// TwinCAT 3 PLC project MqttTestPLC2
// ProgramVersion: 3.1.4023.0
// libraries:
//   ChainControllerLib, * (FactoryAutomation)
//   MqttFramework, * (FactoryAutomation)
//   StateMachineLib, * (FactoryAutomation)
//   StepWorkerLib, * (FactoryAutomation)
//   Tc2_Standard, * (Beckhoff Automation GmbH)
//   Tc2_System, * (Beckhoff Automation GmbH)
//   Tc3_Module, * (Beckhoff Automation GmbH)
// project tree:
//   / PlcTask.TcTTO
//   POUs/Basic/Conveyors/ BeltConveyor.TcPOU, Conveyor.TcPOU, PalletizerConveyor.TcPOU, RollerConveyor.TcPOU
//   POUs/Basic/Cylinder/ Cylinder.TcPOU
//   POUs/Basic/Elevator/ Elevator.TcPOU, PalletizerElevator.TcPOU
//   POUs/Basic/Sensor/ Sensor.TcPOU
//   POUs/HeavyModules/LineRegulator/ SM_LineRegulator.TcPOU
//   POUs/HeavyModules/TransferLine/ SM_TransferLine.TcPOU, TL_BUSY.TcDUT, TL_RollerConveyors.TcDUT
//   POUs/HeavyModules/TransferLine/StepChains/BeltConveyors/ SC_ACTUATOR_BeltConveyors.TcDUT, SC_BeltConveyors.TcPOU, SC_BUSY_BeltConveyors.TcDUT, SC_SENSOR_BeltConveyors.TcDUT
//   POUs/HeavyModules/TransferLine/StepChains/PostPalletizer/ SC_PostPalletizer.TcPOU
//   POUs/HeavyModules/TransferLine/StepChains/PrePalletizer/ SC_PrePalletizer.TcPOU
//   POUs/LightModules/PresenceDetector/ PresenceDetector.TcPOU
//   POUs/LightModules/Turntable/ Turntable.TcPOU
//   POUs/Main/ MAIN.TcPOU, MAIN_BUSY.TcDUT
//   POUs/MediumModules/Palletizer/ PAL_Busy.TcDUT, SM_Palletizer.TcPOU
//   POUs/MediumModules/Palletizer/StepChains/FirstFloor/ SC_BUSY_FirstFloor.TcDUT, SC_FirstFloor.TcPOU
//   POUs/MediumModules/Palletizer/StepChains/SecondFloor/ SC_BUSY_SecondFloor.TcDUT, SC_SecondFloor.TcPOU
//   VISUs/ Visu.TcPOU
// real-time tasks:
//   TASK PlcTask: cycle T#10ms, priority 21, ADS port 350

CONFIGURATION MqttTestPLC2
    RESOURCE PLC ON TwinCAT3
        TASK PlcTask(INTERVAL := T#10ms, PRIORITY := 21);
        PROGRAM MAIN WITH PlcTask : MAIN;
        PROGRAM ADS WITH PlcTask : ADS;
    END_RESOURCE
END_CONFIGURATION

// ---- POUs/HeavyModules/TransferLine/StepChains/BeltConveyors/SC_ACTUATOR_BeltConveyors.TcDUT

TYPE SC_ACTUATOR_BeltConveyors :
(
	eBeltConveyorEntrance := 1,
	eBeltConveyorUpwards,
	eMaxNumBeltConveyors
)UINT;
END_TYPE

// ---- POUs/HeavyModules/TransferLine/StepChains/BeltConveyors/SC_BUSY_BeltConveyors.TcDUT

TYPE SC_BUSY_BeltConveyors :
(
	eBusySCStart := 0,
	eStartEntranceConveyor,
	eStartUpwardsConveyor,
	eExecutePalletizer,
	eStopEntranceConveyor,
	eWaitForPalletizer,
	eSignalError
)UINT;
END_TYPE

// ---- POUs/HeavyModules/TransferLine/StepChains/BeltConveyors/SC_SENSOR_BeltConveyors.TcDUT

TYPE SC_SENSOR_BeltConveyors :
(
	eCounterSensor := 1,
	eBeltConveyorsMaxSensors
)UINT;
END_TYPE

// ---- POUs/HeavyModules/TransferLine/TL_BUSY.TcDUT

TYPE TL_BUSY :
(
	eTlStartUnits := 0,
	eTlCheckUnits,
	eTlSignalError
)UINT;
END_TYPE

// ---- POUs/HeavyModules/TransferLine/TL_RollerConveyors.TcDUT

TYPE TL_RollerConveyors :
(
	eRollerConveyorEntrance := 1,
	eRollerConveyorExit,
	eRollerConveyorPrePalletizer,
	eTlMaxNumRollerConveyors
)UINT;
END_TYPE

// ---- POUs/Main/MAIN_BUSY.TcDUT

TYPE MAIN_BUSY :
(
	eMainWaitStart := 0
);
END_TYPE

// ---- POUs/MediumModules/Palletizer/PAL_Busy.TcDUT

TYPE PAL_Busy :
(
	ePALStart := 0
	
	
);
END_TYPE

// ---- POUs/MediumModules/Palletizer/StepChains/FirstFloor/SC_BUSY_FirstFloor.TcDUT

TYPE SC_BUSY_FirstFloor :
(
	enum_member := 0
);
END_TYPE

// ---- POUs/MediumModules/Palletizer/StepChains/SecondFloor/SC_BUSY_SecondFloor.TcDUT

TYPE SC_BUSY_SecondFloor :
(
	eSecondFloorStart := 0,
	eActivateTurn,
	eActivateBeltForw,
	eWaitForPackages,
	ePushPackages,
	eRetractPusher,
	eClamp,
	eRetractClamper,
	eWaitForPallet,
	eOpenPlate,
	eClosePlate,
	eElevatorUp,
	eElevatorDown,
	eStartChains,
	eStopChains,
	eWaitForFirstFloor,
	eSyncWithFirstFloor,
	eSecondFloorDone
);
END_TYPE

// ---- POUs/Main/MAIN.TcPOU
PROGRAM MAIN
VAR
 
 fbLineRegulator : SM_LineRegulator;
 fbSymbolPathStorage : SymbolPathStorage;

END_VAR

fbLineRegulator(
	 sSubscription1 := 'TL1Synch',
	 sSubscription2 := 'TL2Synch',
	 sSubscription3 := 'TL3Synch'
);

END_PROGRAM

// ---- POUs/HeavyModules/LineRegulator/SM_LineRegulator.TcPOU
FUNCTION_BLOCK SM_LineRegulator EXTENDS StateMachine
VAR_INPUT
	 sSubscription1 : STRING(8);
	 sSubscription2 : STRING(8);
	 sSubscription3 : STRING(8);
END_VAR
VAR_OUTPUT
END_VAR
VAR
	fbTurntable : Turntable;

	aRollerConveyors : ARRAY[1..3] OF RollerConveyor;
	fbRollerConveyorExit : RollerConveyor;
	fbReadyStepWorker : FB_StepWorker;
	fbBusyStepWorker : FB_StepWorker;
	fbInitStepWorker : FB_StepWorker;
	
	messageIndex : UINT;
	stMqttPayload : ST_MqttPayload;
	aSubscriptions : ARRAY[1..3] OF STRING(8);
	uiSubscriptionsCycler : UINT := 1;
END_VAR

SUPER^();
fbTurntable();
aRollerConveyors[1]();
aRollerConveyors[3]();

METHOD PROTECTED   Busy : BOOL
VAR_INPUT
END_VAR
fbBusyStepWorker();
CASE fbBusyStepWorker.uiStep OF

	0:
	
		aRollerConveyors[uiSubscriptionsCycler].On();
		CASE uiSubscriptionsCycler OF
		
			1:
				fbTurntable.RollMinus();
				fbTurntable.Turn();
			
			2:
				fbTurntable.RollPlus();
			
			3:
				fbTurntable.RollPlus();
				fbTurntable.Turn();
		END_CASE
		
		fbBusyStepWorker
			.mAddCondition(itfStepCondition := fbTurntable.fbBackLimit.getSignal)
			.mNextStep(10);
			
	10:
	
		aRollerConveyors[uiSubscriptionsCycler].Off();
		CASE uiSubscriptionsCycler OF
		
			1:
				fbTurntable.StopRolling();			
				fbTurntable.UnTurn();
				fbBusyStepWorker
					.mSetTimer(T#2S)
					.mNextStep(20);
			
			2:
				fbBusyStepWorker.mNextStep(30);
			
			3:
				fbTurntable.StopRolling();
				fbTurntable.UnTurn();
				fbBusyStepWorker
					.mSetTimer(T#2S)
					.mNextStep(20);
		END_CASE
		
	20:
	
		fbTurntable.RollPlus();
		fbRollerConveyorExit.On();
		fbBusyStepWorker
			.mSetTimer(T#10S)
			.mNextStep(30);
	30:	
	
		IF NOT fbTurntable.fbBackLimit.bSignal
			AND NOT fbTurntable.fbFrontLimit.bSignal
		THEN
			fbRollerConveyorExit.Off();
			fbBusyStepWorker
				.mSetTimer(T#1S)
				.mNextStep(40);
		END_IF
		
	40:
	
		fbBusyStepWorker.mNextStep(0);
		Done();
		
	
END_CASE
END_METHOD

METHOD PROTECTED  Error : BOOL
VAR_INPUT
END_VAR
END_METHOD

METHOD PROTECTED  Idle : BOOL
VAR_INPUT
END_VAR
END_METHOD

METHOD PROTECTED  Init : BOOL
VAR_INPUT
END_VAR
fbInitStepWorker();
CASE fbInitStepWorker.uiStep OF

	0: 
	
		IF ADS.fbAdsConnector.isConnected
		THEN
			fbInitStepWorker.mNextStep(10);
		END_IF
		
	10:
	
		IF ADS.fbMqttClient.Subscribe(sSubscription1)
		THEN			
			fbInitStepWorker.mNextStep(20);
		END_IF
		
	20:
	
		IF ADS.fbMqttClient.Subscribe(sSubscription2)
		THEN			
			fbInitStepWorker.mNextStep(30);
		END_IF
		
	30:
		
		IF ADS.fbMqttClient.Subscribe(sSubscription3)
		THEN		
			aSubscriptions[1] := sSubscription1;
			aSubscriptions[2] := sSubscription2;
			aSubscriptions[3] := sSubscription3;
			Start();
		END_IF		
		
END_CASE
END_METHOD

METHOD PROTECTED  Prepare : BOOL
VAR_INPUT
END_VAR
END_METHOD

METHOD PROTECTED  Ready : BOOL
VAR_INPUT
END_VAR
VAR
	
END_VAR
fbReadyStepWorker();


CASE fbReadyStepWorker.uiStep OF

	0: 
		IF NOT fbTurntable.bBackLimit
			AND NOT fbTurntable.bFrontLimit
		THEN
			fbReadyStepWorker.mNextStep(10);
		END_IF
		
	10:
	
		IF uiSubscriptionsCycler = 3
		THEN
			uiSubscriptionsCycler := 1;
		ELSE
			uiSubscriptionsCycler := uiSubscriptionsCycler + 1;
		END_IF
		
		messageIndex := ADS.fbMqttClient.isNewMessage(aSubscriptions[uiSubscriptionsCycler]);
		IF messageIndex > 0
		THEN
			stMqttPayload := Ads.fbMqttClient.getNewMessage(messageIndex);
			fbReadyStepWorker.mNextStep(20);
		END_IF
		
	20:	
		Ads.fbMqttClient.Publish(aSubscriptions[uiSubscriptionsCycler],stMqttPayload);
		fbReadyStepWorker.mNextStep(0);
		Execute();
		
END_CASE
END_METHOD

METHOD PROTECTED  Waiting : BOOL
VAR_INPUT
END_VAR
END_METHOD

END_FUNCTION_BLOCK

// ---- POUs/LightModules/Turntable/Turntable.TcPOU
FUNCTION_BLOCK Turntable
VAR_INPUT



END_VAR
VAR_OUTPUT

	bTurn 		: BOOL;
	bRollPlus	: BOOL;
	bRollMinus 	: BOOL;
	bFrontLimit : BOOL;
	bBackLimit	: BOOL;
	
END_VAR
VAR

	fbFrontLimit : Sensor;
	fbBackLimit : Sensor;
	
	fbTurn : BoolOut;
	fbRollPlus : BoolOut;
	fbRollMinus : BoolOut;
	
END_VAR

fbFrontLimit();
fbBackLimit();

bTurn := fbTurn.getValue;
bRollPlus := fbRollPlus.getValue;
bRollMinus := fbRollMinus.getValue;
bFrontLimit := fbFrontLimit.bSignal;
bBackLimit	:= fbBackLimit.bSignal;

METHOD RollMinus : BOOL
VAR_INPUT
END_VAR
fbRollMinus.setValue := TRUE;
fbRollPlus.setValue := FALSE;
END_METHOD

METHOD RollPlus : BOOL
VAR_INPUT
END_VAR
fbRollPlus.setValue := TRUE;
fbRollMinus.setValue := FALSE;
END_METHOD

METHOD StopRolling : BOOL
VAR_INPUT
END_VAR
fbRollMinus.setValue := FALSE;
fbRollPlus.setValue := FALSE;
END_METHOD

METHOD Turn : BOOL
VAR_INPUT
END_VAR
fbTurn.setValue := TRUE;
END_METHOD

METHOD Unturn : BOOL
VAR_INPUT
END_VAR
fbTurn.setValue := FALSE;
END_METHOD

END_FUNCTION_BLOCK

// ---- POUs/Basic/Sensor/Sensor.TcPOU
FUNCTION_BLOCK Sensor
VAR_INPUT
END_VAR
VAR_OUTPUT
	bSignal  : BOOL;
END_VAR
VAR
	fbSignal : BoolIn;
END_VAR

bSignal := fbSignal.getValue;

PROPERTY getSignal : I_StepCondition
GET
getSignal := fbSignal;
END_GET
END_PROPERTY

END_FUNCTION_BLOCK

// ---- POUs/Basic/Conveyors/RollerConveyor.TcPOU
FUNCTION_BLOCK RollerConveyor EXTENDS Conveyor
VAR_INPUT
END_VAR
VAR_OUTPUT
END_VAR
VAR
END_VAR

Super^();

END_FUNCTION_BLOCK

// ---- POUs/Basic/Conveyors/Conveyor.TcPOU
FUNCTION_BLOCK Conveyor 
VAR_INPUT
END_VAR

VAR_OUTPUT
	bStart  : BOOL;
END_VAR
VAR
	fbStart : BoolOut;
END_VAR

bStart := fbStart.getValue;

PROPERTY getStart : I_StepCondition
GET
getStart := fbStart;
END_GET
END_PROPERTY

METHOD Off : BOOL
VAR_INPUT
END_VAR
fbStart.setValue := FALSE;
END_METHOD

METHOD On : BOOL
VAR_INPUT
END_VAR
fbStart.setValue := TRUE;
END_METHOD

END_FUNCTION_BLOCK

// ---- POUs/Basic/Conveyors/BeltConveyor.TcPOU
FUNCTION_BLOCK BeltConveyor EXTENDS Conveyor
VAR_INPUT
END_VAR
VAR_OUTPUT
END_VAR
VAR
END_VAR

Super^();

END_FUNCTION_BLOCK

// ---- POUs/Basic/Conveyors/PalletizerConveyor.TcPOU
FUNCTION_BLOCK PalletizerConveyor EXTENDS Conveyor
VAR_INPUT
END_VAR
VAR_OUTPUT
	bStartBackward : BOOL;
END_VAR
VAR	
	fbStartBackward : BoolOut;
END_VAR

SUPER^();
bStartBackward := fbStartBackward.getValue;

PROPERTY getStartBackward : I_StepCondition
GET
getStartBackward := fbStartBackward;
END_GET
END_PROPERTY

END_FUNCTION_BLOCK

// ---- POUs/Basic/Cylinder/Cylinder.TcPOU
FUNCTION_BLOCK Cylinder 
VAR_INPUT
END_VAR
VAR_OUTPUT
	bExtended : BOOL;
	bExtend : BOOL;
END_VAR
VAR
	fbExtendedSignal : BoolIn;
	fbExtend : BoolOut;
END_VAR

bExtended := fbExtendedSignal.getValue;
bExtend := fbExtend.getValue;

METHOD Extend : BOOL
VAR_INPUT
END_VAR
fbExtend.setValue := TRUE;
END_METHOD

PROPERTY getExtend : I_StepCondition
GET
getExtend := fbExtend;
END_GET
END_PROPERTY

METHOD Retract : BOOL
VAR_INPUT
END_VAR
fbExtend.setValue := FALSE;
END_METHOD

END_FUNCTION_BLOCK

// ---- POUs/Basic/Elevator/Elevator.TcPOU
FUNCTION_BLOCK Elevator
VAR_INPUT
END_VAR
VAR_OUTPUT
END_VAR
VAR
END_VAR

END_FUNCTION_BLOCK

// ---- POUs/Basic/Elevator/PalletizerElevator.TcPOU
FUNCTION_BLOCK PalletizerElevator EXTENDS Elevator
VAR_INPUT
END_VAR
VAR_OUTPUT
	isMoving : BOOL;
END_VAR
VAR
	fbElevatorMoving : Sensor;
	fbElevatorUp : BoolOut;
	fbElevatorDown : BoolOut;
	fbElevatorToLimit : BoolOut;
END_VAR

isMoving := fbElevatorMoving.bSignal;

PROPERTY getElevatorMoving : I_StepCondition
GET
getElevatorMoving := fbElevatorMoving.getSignal;
END_GET
END_PROPERTY

METHOD MoveDown : BOOL
VAR_INPUT
END_VAR
fbElevatorDown.setValue := TRUE;
fbElevatorUp.setValue := FALSE;

fbElevatorToLimit.setValue := TRUE;
END_METHOD

METHOD MoveUp : BOOL
VAR_INPUT
END_VAR
fbElevatorUp.setValue := TRUE;
fbElevatorDown.setValue := FALSE;

fbElevatorToLimit.setValue := TRUE;
END_METHOD

END_FUNCTION_BLOCK

// ---- POUs/HeavyModules/TransferLine/SM_TransferLine.TcPOU
FUNCTION_BLOCK SM_TransferLine EXTENDS StateMachine
VAR_INPUT CONSTANT
	sTLMqttName : STRING(8);
END_VAR
VAR_OUTPUT
END_VAR
VAR
	
	aRollerConveyors : ARRAY[1..3] OF RollerConveyor;
	fbChainController : FB_ChainController;
	
	fbPalletizer : SM_Palletizer;
	fbStepWorkerReady : FB_StepWorker;
	fbStepWorkerBusy : FB_StepWorker;

	scBeltConveyors : 
		SC_BeltConveyors := 
		(
			sChainName  := 'scBeltConveyors',
			rChainController := fbChainController
		);
		
	scPostPalletizer : 
		SC_PostPalletizer := 
		(
			sChainName  := 'scPostPalletizer',
			rChainController := fbChainController
		);
		
	scPrePalletizer : 
		SC_PrePalletizer := 
		(
			sChainName  := 'scPrePalletizer',
			rChainController := fbChainController
		);
 
	uiPackageCounter : UINT;
	i : UINT;
	bPackageOnTheWay : BOOL;
	
END_VAR

SUPER^();
fbPalletizer(ioChainController := fbChainController);
scBeltConveyors(bAllPartsPresent := fbPalletizer.bAllPartsPresent);
scPrePalletizer();
scPrePalletizer.bPalletizerRequest := fbPalletizer.scFirstFloor.bPalletizerRequest;
fbPalletizer.scFirstFloor.bIncomingPallet := scPrePalletizer.bSentToPalletizer;
scPostPalletizer(sTLMqttName := sTLMqttName);

METHOD PROTECTED Busy : BOOL
VAR_INPUT
END_VAR
CASE fbStepWorkerBusy.uiStep OF
	eTlStartUnits:
		scBeltConveyors.bExecute := TRUE;
		scPrePalletizer.bExecute := TRUE;
		scPostPalletizer.bExecute := TRUE;
		fbPalletizer.bExecute := TRUE;
		fbStepWorkerBusy.mNextStep(eTlCheckUnits);
	eTlCheckUnits:
		IF scBeltConveyors.eStateMachine = E_StateMachine.eError
		THEN
			fbStepWorkerBusy.mNextStep(eTlSignalError);
		END_IF
	eTlSignalError:
		Fault();
END_CASE
END_METHOD

METHOD PROTECTED  Error : BOOL
VAR_INPUT
END_VAR
END_METHOD

METHOD PROTECTED  Idle : BOOL
VAR_INPUT
END_VAR
Start();
END_METHOD

METHOD PROTECTED  Init : BOOL
VAR_INPUT
END_VAR
fbChainController
	.addChain(itfChain := scBeltConveyors)
	.addChain(itfChain := scPostPalletizer)
	.addChain(itfChain := scPrePalletizer);
	
	
Start();
END_METHOD

METHOD PROTECTED  Prepare : BOOL
VAR_INPUT
END_VAR
END_METHOD

METHOD PROTECTED  Ready : BOOL
VAR_INPUT
END_VAR
END_METHOD

METHOD PROTECTED  Waiting : BOOL
VAR_INPUT
END_VAR
END_METHOD

END_FUNCTION_BLOCK

// ---- POUs/MediumModules/Palletizer/SM_Palletizer.TcPOU
FUNCTION_BLOCK SM_Palletizer EXTENDS StateMachine
VAR_INPUT
	bExecute : BOOL;
	scFirstFloor : SC_FirstFloor;	
	scSecondFloor : SC_SecondFloor;
END_VAR
VAR_IN_OUT
	ioChainController : FB_ChainController;
END_VAR
VAR_OUTPUT
	
	bAllPartsPresent: BOOL;	
	
END_VAR
VAR

	fbDoneCycle : BoolOut;
	fbStepWorkerBusy : FB_StepWorker;
	
	
END_VAR

SUPER^();
scFirstFloor(bExecute := bExecute);
scSecondFloor(bExecute := bExecute);

bAllPartsPresent := scSecondFloor.bAllPartsPresent;
scSecondFloor.bPlateOpen := scFirstFloor.bPlateOpen;

METHOD PROTECTED   Busy : BOOL
VAR_INPUT
END_VAR
scFirstFloor(bExecute := TRUE);
scSecondFloor(bExecute := TRUE);
END_METHOD

METHOD PROTECTED  Error : BOOL
VAR_INPUT
END_VAR
END_METHOD

PROPERTY getDoneCycle : I_StepCondition
GET
getDoneCycle := fbDoneCycle;
END_GET
END_PROPERTY

METHOD PROTECTED  Idle : BOOL
VAR_INPUT
END_VAR
Start();
END_METHOD

METHOD PROTECTED  Init : BOOL
VAR_INPUT
END_VAR
ioChainController
	.addChain(itfChain := scFirstFloor)
	.addChain(itfChain := scSecondFloor);
	
scFirstFloor(
	sChainName := 'scFirstFloor',
	rChainController := ioChainController
);
scSecondFloor(
	sChainName := 'scSecondFloor',
	rChainController := ioChainController
);
Start();
END_METHOD

METHOD PROTECTED  Prepare : BOOL
VAR_INPUT
END_VAR
END_METHOD

METHOD PROTECTED  Ready : BOOL
VAR_INPUT
END_VAR
END_METHOD

METHOD PROTECTED  Waiting : BOOL
VAR_INPUT
END_VAR
END_METHOD

END_FUNCTION_BLOCK

// ---- POUs/MediumModules/Palletizer/StepChains/FirstFloor/SC_FirstFloor.TcPOU
FUNCTION_BLOCK SC_FirstFloor EXTENDS FB_Chain
VAR_INPUT
	bExecute : BOOL;
	bIncomingPallet : BOOL;
	bPostPalletizerRequestGranted : BOOL;
END_VAR
VAR_OUTPUT
	bPlateOpen : BOOL;
	bPalletizerRequest : BOOL;
	bSentToPostPalletizer : BOOL;
	bPostPalletizerDeliveryRequest : BOOL;
END_VAR
VAR
	fbPallChainConveyor : PalletizerConveyor;
	fbPallElevator : PalletizerElevator;
	fbPlateCyl : Cylinder;
	fbPlateLimitSen : Sensor;
	fbElevatorFrontLimit : Sensor;
	fbElevatorBackLimit : Sensor;
END_VAR

SUPER^();
bPlateOpen := fbPlateCyl.bExtended;
fbPallChainConveyor();
fbPallElevator();
fbPlateCyl();
fbPlateLimitSen();

METHOD PROTECTED   Busy : BOOL
VAR_INPUT
END_VAR

		
fbStepWorkerBusy();
CASE fbStepWorkerBusy.uiStep OF
	
	0: 
		fbPallChainConveyor.On();
		fbStepWorkerBusy
			.mAddCondition(itfStepCondition := fbElevatorBackLimit.getSignal)
			.mAddCondition(itfStepCOndition := fbElevatorFrontLimit.getSignal)
			.mNextStep(10);
			
	10: 
	
		fbPallChainConveyor.Off();
		bPalletizerRequest := FALSE;
		IF rChainController
			.releaseCheck(THIS^)
			.releaseFromChain(sChainReleasing := 'scSecondFloor', THIS^)
			.releaseResult(THIS^) 
		THEN
			fbStepWorkerBusy.mNextStep(20);
		END_IF

	20:
	
		fbPallElevator.MoveUp();
		fbStepWorkerBusy
			.mSetTimer(T#1S)
			.mNextStep(30);
			
	30:
	
		IF NOT fbPallElevator.isMoving
		THEN
			fbStepWorkerBusy
				.mSetTimer(tTime := T#2S)
				.mNextStep(40);
		END_IF
		
	40:
	
		fbPlateCyl.Extend();
		fbStepWorkerBusy
			.mSetTimer(T#2S)
			.mNextStep(45);
	
	45:	
		rChainController.releaseForChain('scSecondFloor', THIS^);	
		fbPallElevator.MoveDown();		
		fbStepWorkerBusy
			.mSetTimer(T#2S)
			.mNextStep(50);
	50:
	
		IF NOT fbPallElevator.isMoving
		THEN
			rChainController.releaseForChain('scPostPalletizer', THIS^);
			fbStepWorkerBusy.mNextStep(60);
		END_IF
	
		
	60:
	
		fbPlateCyl.Retract();
		fbStepWorkerBusy.mNextStep(100);
	
	100:
	
		IF rChainController
			.releaseCheck(THIS^)
			.releaseFromChain(sChainReleasing := 'scPostPalletizer', THIS^)
			.releaseResult(THIS^) 
		THEN

			fbPallChainConveyor.On();
			fbStepWorkerBusy.mNextStep(105);
			
		END_IF

	105:
		fbStepWorkerBusy
				.mSetTimer(T#2s)
				.mNextStep(110);
	110:		
		
		IF NOT fbElevatorBackLimit.bSignal
			AND NOT fbElevatorFrontLimit.bSignal
		THEN
		
			Done();
			fbPallChainConveyor.Off();
			fbStepWorkerBusy.mNextStep(0);
		END_IF

END_CASE
END_METHOD

METHOD PROTECTED  Error : BOOL
VAR_INPUT
END_VAR
END_METHOD

METHOD PROTECTED  Idle : BOOL
VAR_INPUT
END_VAR
END_METHOD

METHOD PROTECTED  Init : BOOL
VAR_INPUT
END_VAR
Start();
END_METHOD

METHOD PROTECTED  Prepare : BOOL
VAR_INPUT
END_VAR
END_METHOD

METHOD PROTECTED  Ready : BOOL
VAR_INPUT
END_VAR

fbStepWorkerReady();
CASE fbStepWorkerReady.uiStep OF
	
	0: 
	
		IF bExecute THEN
			fbStepWorkerReady.mNextStep(10);
		END_IF
		
	10:

		IF NOT fbElevatorFrontLimit.bSignal
			AND NOT fbElevatorBackLimit.bSignal 
		THEN
			bPalletizerRequest := TRUE;
			fbStepWorkerReady.mNextStep(20);
		END_IF
		
	20:
	
		IF bIncomingPallet
		THEN
			fbStepWorkerReady.mNextStep(0);
			Execute();
		END_IF
		
		
END_CASE
END_METHOD

METHOD PROTECTED  Waiting : BOOL
VAR_INPUT
END_VAR
END_METHOD

END_FUNCTION_BLOCK

// ---- POUs/MediumModules/Palletizer/StepChains/SecondFloor/SC_SecondFloor.TcPOU
FUNCTION_BLOCK SC_SecondFloor EXTENDS FB_Chain
VAR_INPUT
	bExecute : BOOL;
	bPlateOpen : BOOL;
END_VAR
VAR_OUTPUT
	bAllPartsPresent: BOOL;	
END_VAR
VAR
	fbPallBeltConveyor : PalletizerConveyor;
	fbPushCyl : Cylinder;
	fbTurnCyl : Cylinder;
	
	fbClampCyl : Cylinder;
	fbClampedSen : Sensor;
	
	fbPusherLimitSen : Sensor;
	fbPresenceDetector : PresenceDetector;
	iCycle : INT;
END_VAR

SUPER^();

fbPushCyl();
fbTurnCyl();

fbClampCyl();
fbPallBeltConveyor();
fbPresenceDetector(bAllPartsPresent => bAllPartsPresent);

METHOD PROTECTED   Busy : BOOL
VAR_INPUT
END_VAR
fbStepWorkerBusy();
CASE fbStepWorkerBusy.uiStep OF
	
	eSecondFloorStart: //send release to scBeltConveyor
	
		iCycle := iCycle + 1;
		IF iCycle = 2
		THEN
			rChainController.releaseForChain('scBeltConveyors', THIS^);
			fbStepWorkerBusy.mNextStep(10);
		ELSE
			fbStepWorkerBusy.mNextStep(20);
		END_IF
		
		
		
	10: //wait for release from scBeltConveyor to start actuators
	
		IF rChainController
			.releaseCheck(THIS^)
			.releaseFromChain(sChainReleasing := 'scBeltConveyors', THIS^)
			.releaseResult(THIS^) 
		THEN
			fbStepWorkerBusy.mNextStep(20);
		END_IF
	
		
	20: //wait for packages
		
		fbTurnCyl.Extend();
		fbPallBeltConveyor.On();
		IF fbPresenceDetector.bAllPartsPresent
		THEN
			bAllPartsPresent := TRUE;
			fbPallBeltConveyor.Off();
			fbStepWorkerBusy.mNextStep(ePushPackages);
		END_IF	
		
	ePushPackages:
	
		fbPushCyl.Extend();
		
		fbStepWorkerBusy
			.mSetTimer(T#2S)
			.mNextStep(eRetractPusher);
		
	eRetractPusher:
	
		fbPushCyl.Retract();
		
		fbStepWorkerBusy
			.mSetTimer(T#2S)
			.mNextStep(eClamp);
			
	eClamp:
	
		fbClampCyl.Extend();
		fbStepWorkerBusy
			.mSetTimer(T#2S)
			.mNextStep(eRetractClamper);
			
	eRetractClamper:
	
		
		fbClampCyl.Retract();
		IF iCycle = 1
		THEN
			fbStepWorkerBusy
				.mSetTimer(T#2S)
				.mNextStep(eSecondFloorStart);
		ELSE
			iCycle := 0;
			fbStepWorkerBusy.mNextStep(eSyncWithFirstFloor);
		END_IF
		
	eSyncWithFirstFloor:
	
		rChainController.releaseForChain('scFirstFloor', THIS^);	
		fbStepWorkerBusy.mNextStep(eWaitForFirstFloor);
	
	eWaitForFirstFloor:
	
		IF rChainController
			.releaseCheck(THIS^)
			.releaseFromChain(sChainReleasing := 'scFirstFloor', THIS^)
			.releaseResult(THIS^) 
		THEN
			fbStepWorkerBusy.mNextStep(eSecondFloorDone);
		END_IF
		
	eSecondFloorDone:
		fbStepWorkerBusy.mNextStep(eSecondFloorStart);
		Done();	
	
END_CASE
END_METHOD

METHOD PROTECTED  Error : BOOL
VAR_INPUT
END_VAR
END_METHOD

METHOD PROTECTED  Idle : BOOL
VAR_INPUT
END_VAR
END_METHOD

METHOD PROTECTED  Init : BOOL
VAR_INPUT
END_VAR
Start();
END_METHOD

METHOD PROTECTED  Prepare : BOOL
VAR_INPUT
END_VAR
END_METHOD

METHOD PROTECTED  Ready : BOOL
VAR_INPUT
END_VAR

fbStepWorkerReady();
CASE fbStepWorkerReady.uiStep OF
	
	0: 
	
		IF bExecute THEN
			fbStepWorkerReady.mNextStep(10);
		END_IF
		
	10:
		
		IF NOT fbPresenceDetector.bAllPartsPresent
			AND NOT bPlateOpen
		THEN
			rChainController.releaseForChain('scBeltConveyors', THIS^);	
			fbStepWorkerReady.mNextStep(20);	
		END_IF
	
	20:
		
		IF rChainController
			.releaseCheck(THIS^)
			.releaseFromChain(sChainReleasing := 'scBeltConveyors', THIS^)
			.releaseResult(THIS^) 
		THEN
			fbStepWorkerReady.mNextStep(0);
			Execute();
		END_IF
		
END_CASE
END_METHOD

METHOD PROTECTED  Waiting : BOOL
VAR_INPUT
END_VAR
END_METHOD

END_FUNCTION_BLOCK

// ---- POUs/LightModules/PresenceDetector/PresenceDetector.TcPOU
FUNCTION_BLOCK PresenceDetector
VAR_INPUT
END_VAR
VAR_OUTPUT
	bAllPartsPresent : BOOL;
END_VAR
VAR
	aSensors : ARRAY[1..3] OF Sensor;
	fbTimer : TON;
	i: INT;
END_VAR

aSensors[1]();
aSensors[2]();
aSensors[3]();
fbTimer(
	IN:= aSensors[1].bSignal
		AND aSensors[2].bSignal
		AND aSensors[3].bSignal,
	PT:=T#2S
);
IF fbTimer.Q
THEN
	bAllPartsPresent := TRUE;
ELSE
	bAllPartsPresent :=FALSE;
END_IF

END_FUNCTION_BLOCK

// ---- POUs/HeavyModules/TransferLine/StepChains/BeltConveyors/SC_BeltConveyors.TcPOU
FUNCTION_BLOCK SC_BeltConveyors EXTENDS FB_Chain
VAR_INPUT
	bExecute : BOOL;
	bAllPartsPresent : BOOL;
END_VAR
VAR_OUTPUT
END_VAR
VAR
	aBeltConveyors : ARRAY[1..2] OF BeltConveyor;
	fbCounterSensor : Sensor;
	i : INT;
	uiPackageCounter : UINT;
	fbTrig : R_TRIG;
	
END_VAR

SUPER^();
fbCounterSensor();
fbTrig(CLK := fbCounterSensor.bSignal);
IF fbTrig.Q
THEN
	uiPackageCounter := uiPackageCounter + 1;
END_IF
FOR i := 1 TO (eMaxNumBeltConveyors - 1)
DO
	
	aBeltConveyors[i]();

END_FOR

METHOD PROTECTED Busy : BOOL
VAR_INPUT
END_VAR
VAR
	iStepCondition : I_StepCondition;
END_VAR
fbStepWorkerBusy();

CASE fbStepWorkerBusy.uiStep OF

	eBusySCStart: 
		THIS^.aBeltConveyors[eBeltConveyorEntrance].On();
		
		fbStepWorkerBusy.mNextStep(10);
		
	10:
		//As Soon as the first package reaches the counter sensor
		//the second floor of the palletizer is informed
		//consequently the second floor of the palletizer will go in busy mode.
		IF uiPackageCounter = 1
		THEN
			THIS^.aBeltConveyors[eBeltConveyorUpwards].On();
			
			fbStepWorkerBusy.mNextStep(15);
		END_IF
		
	15:
		IF uiPackageCounter = 3
		THEN
			uiPackageCounter := 0;
			fbStepWorkerBusy.mNextStep(20);
		END_IF
	20:
		fbStepWorkerBusy
				.mSetTimer(T#1s)
				.mNextStep(30);
	30:
		THIS^.aBeltConveyors[eBeltConveyorEntrance].Off();
		IF bAllPartsPresent
		THEN
			THIS^.aBeltConveyors[eBeltConveyorUpwards].Off();
			Done();
			fbStepWorkerBusy.mNextStep(0);
		END_IF
		
	40:
	
		
		(*
		//At start we check how many packages have passed the fbCounterSensor
		IF uiPackageCounter < 3
		THEN
		
			//activate the conveyors
			fbStepWorkerBusy.mNextStep(eStartEntranceConveyor);
			
		ELSIF uiPackageCounter = 3
		 AND NOT ioPalletizer.bAllPartsPresent
		 AND aBeltConveyors[eBeltConveyorEntrance].bStart
		THEN
 			//A package needs to reach the palletizer or a sensor is malfunctioning		
			fbStepWorkerBusy
				.mSetTimer(T#1s)
				.mNextStep(eStopEntranceConveyor);
				
		ELSIF uiPackageCounter = 3
		 AND ioPalletizer.bAllPartsPresent
	 	THEN
			//Execute the Palletizer
			uiPackageCounter := 0;
			aBeltConveyors[eBeltConveyorUpwards].Off();
			fbStepWorkerBusy.mNextStep(eWaitForPalletizer);
		ELSIF uiPackageCounter > 3
		THEN
			//Error
		END_IF
		
	eStartEntranceConveyor:
		
		aBeltConveyors[eBeltConveyorEntrance].On();
		fbStepWorkerBusy.mAddCondition(fbCounterSensor.getSignal);
		fbStepWorkerBusy.mNextStep(eStartUpwardsConveyor);

	eStartUpwardsConveyor:
	
		
		aBeltConveyors[eBeltConveyorUpwards].On();
		fbStepWorkerBusy.mNextStep(eExecutePalletizer);
			 
	eExecutePalletizer:
		 
		ioPalletizer.Execute();	
		fbStepWorkerBusy.mNextStep(eBusySCStart);
	
	eStopEntranceConveyor:
		aBeltConveyors[eBeltConveyorEntrance].Off();
		fbStepWorkerBusy.mNextStep(eExecutePalletizer);
		
	eWaitForPalletizer:
	
		 fbStepWorkerBusy.mAddCondition(ioPalletizer.getDoneCycle);
		 fbStepWorkerBusy.mNextStep(eBusySCStart);
		 
	eSignalError:
	
		fbStepWorkerBusy.mNextStep(eBusySCStart);
		Fault();	
		*)	
END_CASE
END_METHOD

METHOD PROTECTED  Error : BOOL
VAR_INPUT
END_VAR
VAR
	i : INT;
END_VAR
FOR i := 1 TO 3 
DO

	aBeltConveyors[i].Off();
	
END_FOR
END_METHOD

METHOD PROTECTED  Idle : BOOL
VAR_INPUT
END_VAR
END_METHOD

METHOD PROTECTED  Init : BOOL
VAR_INPUT
END_VAR
Start();
END_METHOD

METHOD PROTECTED  Prepare : BOOL
VAR_INPUT
END_VAR
END_METHOD

METHOD PROTECTED  Ready : BOOL
VAR_INPUT
END_VAR
fbStepWorkerReady();
CASE fbStepWorkerReady.uiStep OF
	
	0: 
	
		IF bExecute THEN
			fbStepWorkerReady.mNextStep(10);
		END_IF
		
	10:
	
		IF rChainController
			.releaseCheck(THIS^)
			.releaseFromChain(sChainReleasing := 'scSecondFloor', THIS^)
			.releaseResult(THIS^) 
		THEN
			Execute();
			rChainController.releaseForChain('scSecondFloor', THIS^);		
			fbStepWorkerReady.mNextStep(0);
		END_IF
	
		
	
END_CASE
END_METHOD

METHOD PROTECTED  Waiting : BOOL
VAR_INPUT
END_VAR
END_METHOD

END_FUNCTION_BLOCK

// ---- POUs/HeavyModules/TransferLine/StepChains/PostPalletizer/SC_PostPalletizer.TcPOU
FUNCTION_BLOCK SC_PostPalletizer EXTENDS FB_Chain
VAR_INPUT
	bExecute : BOOL;
	bPalletizerDeliveryRequest : BOOL;
	sTLMqttName : STRING(8);
END_VAR
VAR_OUTPUT
	bGrantDeliveryPermission : BOOL;
END_VAR
VAR
	
	fbPalletAvailable : Sensor;
	fbRollConveyor : RollerConveyor;
	
END_VAR

SUPER^();
fbPalletAvailable();
fbRollConveyor();

METHOD PROTECTED   Busy : BOOL
VAR_INPUT
END_VAR
VAR
	stMqttPayload : ST_MqttPayload;
	messageIndex : UINT;
END_VAR
fbStepWorkerBusy();
CASE fbStepWorkerBusy.uiStep OF
	
	0: 
		THIS^.fbRollConveyor.On();
		rChainController.releaseForChain('scFirstFloor', THIS^);
		fbStepWorkerBusy.mNextStep(10);
		
	10:
		IF THIS^.fbPalletAvailable.bSignal
		THEN
			THIS^.fbRollConveyor.Off();
			fbStepWorkerBusy.mNextStep(20);
		END_IF
	
	20: 
		
		//Mqtt exchange
		IF Ads.fbMqttClient.Publish(sTLMqttName,stMqttPayload)
		THEN
			fbStepWorkerBusy.mNextStep(30);
		END_IF
	
	30:
	
		messageIndex := ADS.fbMqttClient.isNewMessage(sTLMqttName);
		IF messageIndex > 0
		THEN
			stMqttPayload := Ads.fbMqttClient.getNewMessage(messageIndex);
			fbStepWorkerBusy.mNextStep(40);
		END_IF
		
	40:
	
		THIS^.fbRollConveyor.On();
		fbStepWorkerBusy
			.mSetTimer(T#2S)
			.mNextStep(50);
			
	50:
		
		THIS^.fbRollConveyor.Off();
		Done();
		fbStepWorkerBusy.mNextStep(0);
		
END_CASE
END_METHOD

METHOD PROTECTED  Error : BOOL
VAR_INPUT
END_VAR
END_METHOD

METHOD PROTECTED  Idle : BOOL
VAR_INPUT
END_VAR
END_METHOD

METHOD PROTECTED  Init : BOOL
VAR_INPUT
END_VAR
IF ADS.fbMqttClient.Subscribe(sTopic := sTLMqttName)
THEN			
	Start();
END_IF
END_METHOD

METHOD PROTECTED  Prepare : BOOL
VAR_INPUT
END_VAR
END_METHOD

METHOD PROTECTED  Ready : BOOL
VAR_INPUT
END_VAR

fbStepWorkerReady();
CASE fbStepWorkerReady.uiStep OF
	
0:

	IF bExecute
		AND NOT fbPalletAvailable.bSignal
	THEN
		fbStepWorkerReady.mNextStep(10);
	END_IF
		
10:
	IF rChainController
		.releaseCheck(THIS^)
		.releaseFromChain(sChainReleasing := 'scFirstFloor', THIS^)
		.releaseResult(THIS^) 
	THEN
		fbStepWorkerReady.mNextStep(0);
		Execute();
	END_IF
	
END_CASE
END_METHOD

METHOD PROTECTED  Waiting : BOOL
VAR_INPUT
END_VAR
END_METHOD

END_FUNCTION_BLOCK

// ---- POUs/HeavyModules/TransferLine/StepChains/PrePalletizer/SC_PrePalletizer.TcPOU
FUNCTION_BLOCK SC_PrePalletizer EXTENDS FB_Chain
VAR_INPUT
	bPalletizerRequest : BOOL;
	bExecute : BOOL;
END_VAR
VAR_OUTPUT
	bSentToPalletizer : BOOL;
	bPalletAvailable : BOOL;
END_VAR
VAR
	fbRollConvEntrance : RollerConveyor;
	fbRollConvPrePallet : RollerConveyor;
	fbPalletAvailable : Sensor;
END_VAR

SUPER^();
fbPalletAvailable();
bPalletAvailable := fbPalletAvailable.bSignal;

METHOD PROTECTED   Busy : BOOL
VAR_INPUT
END_VAR
fbStepWorkerBusy();
CASE fbStepWorkerBusy.uiStep OF
	
	0: 
		fbRollConvEntrance.On();
		fbRollConvPrePallet.On();
		IF NOT bPalletAvailable
		THEN
			bSentToPalletizer := TRUE;
			fbStepWorkerBusy.mNextStep(10);
		END_IF

	10:
		IF NOT bPalletizerRequest
		THEN
		
			bSentToPalletizer := FALSE;
			fbRollConvPrePallet.Off();
			fbStepWorkerBusy.mNextStep(0);
			
			Done();
			
		ELSIF bPalletAvailable
		THEN
			fbRollConvEntrance.Off();
		END_IF
		
END_CASE
END_METHOD

METHOD PROTECTED  Error : BOOL
VAR_INPUT
END_VAR
END_METHOD

METHOD PROTECTED  Idle : BOOL
VAR_INPUT
END_VAR
END_METHOD

METHOD PROTECTED  Init : BOOL
VAR_INPUT
END_VAR
Start();
END_METHOD

METHOD PROTECTED  Prepare : BOOL
VAR_INPUT
END_VAR
END_METHOD

METHOD PROTECTED  Ready : BOOL
VAR_INPUT
END_VAR

fbStepWorkerReady();
CASE fbStepWorkerReady.uiStep OF
	
	0:
		IF bExecute
		THEN
			fbStepWorkerReady.mNextStep(5);
		END_IF
		
	5: 
		IF NOT bPalletAvailable
		THEN
			fbRollConvEntrance.On();
		ELSIF bPalletAvailable
		THEN
			fbRollConvEntrance.Off();
			fbStepWorkerReady.mNextStep(10);
		END_IF
		
	10:
		IF bPalletizerRequest
		THEN
			fbStepWorkerReady.mNextStep(0);
			Execute();
		END_IF
		
END_CASE
END_METHOD

METHOD PROTECTED  Waiting : BOOL
VAR_INPUT
END_VAR
END_METHOD

END_FUNCTION_BLOCK

// ---- VISUs/Visu.TcPOU
PROGRAM Visu
VAR
	bStartTL1 : BOOL;
	bStartTL2 : BOOL;
	bStartTL3 : BOOL;
END_VAR

END_PROGRAM
